TYPE U_GCSingleProcessStageTimingView :
UNION
	ByName : ST_GCSingleProcessStageTimings;
	ByIndex : ARRAY[1..8] OF ST_GCSingleProcessStageTiming;
END_UNION
END_TYPE

(* stored: Version 1.1.0.1, ProductVersion 3.1.4026.18
   DUT U_GCSingleProcessStageTimingView: Id {39863beb-58d4-4cac-a8f9-a0b6d99fb32a} *)
